VAR_GLOBAL
	InUnloading	:	BOOL;
	PartPresent	:	BOOL;
	LoadingSequenceActive	:	BOOL;
	UnloadingSequenceActive	:	BOOL;
	instStackerCrane	:	FB_StackerCrane_Numerical;
	processStepsLoading	: StackerCraneStepsLoading;	
	processStepsUnloading	: StackerCraneStepsUnloading;
	LiftLowerPartLoadingprocess	:	TON;
	LiftLowerPartUnloadingprocess	:	TON;
END_VAR

(* stored: Version 1.1.0.1
   GVL Warehouse: Id {ca157c31-864b-49ab-96d9-0cfaf46a1877} *)
